# EPICS autosave request: measComp/measCompApp/Db/measCompWaveformDig_settings.req
$(P)$(R)NumPoints
$(P)$(R)FirstChan
$(P)$(R)NumChans
$(P)$(R)Dwell
$(P)$(R)ExtTrigger
$(P)$(R)ExtClock
$(P)$(R)Continuous
$(P)$(R)Retrigger
$(P)$(R)TriggerCount
$(P)$(R)ReadWF.SCAN
